FUNCTION_BLOCK QueryServiceOpcUa (* Query for Services using OPC UA *)
  (* Standard: 61499-2; Description: Copyright (c) 2019 fortiss GmbH This program and the accompanying materials are made available under the terms of the Eclipse Public License 2.0 which is available at https://www.eclipse.org/legal/epl-2.0/ SPDX-License-Identifier: EPL-2.0 *)
  (* Version 1.0, 2019-09-17, Jose Cabral, fortiss GmbH *)
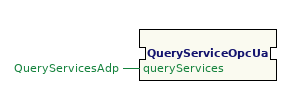
  SOCKETS
    queryServices : QueryServicesAdp;
  END_SOCKETS
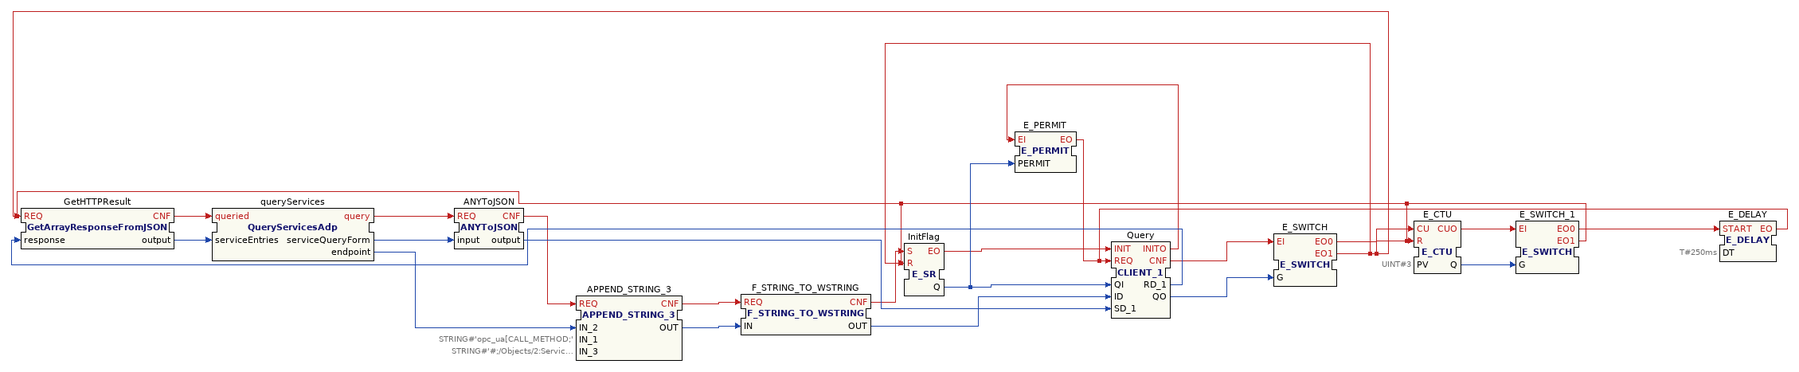
  FBS
    APPEND_STRING_3 : APPEND_STRING_3(IN_1 := STRING#'opc_ua[CALL_METHOD;', IN_3 := STRING#'#;/Objects/2:ServiceRegistry/2:query]');
    F_STRING_TO_WSTRING : F_STRING_TO_WSTRING;
    InitFlag : E_SR;
    E_PERMIT : E_PERMIT;
    ANYToJSON : ANYToJSON;
    GetHTTPResult : GetArrayResponseFromJSON;
    Query : CLIENT_1;
    E_SWITCH_1 : E_SWITCH;
    E_SWITCH : E_SWITCH;
    E_DELAY : E_DELAY(DT := T#250ms);
    E_CTU : E_CTU(PV := UINT#3);
  END_FBS
  EVENT_CONNECTIONS
    APPEND_STRING_3.CNF TO F_STRING_TO_WSTRING.REQ;
    F_STRING_TO_WSTRING.CNF TO InitFlag.S;
    ANYToJSON.CNF TO APPEND_STRING_3.REQ;
    queryServices.query TO ANYToJSON.REQ;
    GetHTTPResult.CNF TO queryServices.queried;
    InitFlag.EO TO Query.INIT;
    E_PERMIT.EO TO Query.REQ;
    Query.INITO TO E_PERMIT.EI;
    E_SWITCH_1.EO0 TO E_DELAY.START;
    E_CTU.CUO TO E_SWITCH_1.EI;
    E_SWITCH.EO0 TO E_CTU.CU;
    E_SWITCH.EO1 TO GetHTTPResult.REQ;
    E_SWITCH.EO1 TO InitFlag.R;
    Query.CNF TO E_SWITCH.EI;
    E_SWITCH_1.EO1 TO InitFlag.R;
    E_SWITCH_1.EO1 TO GetHTTPResult.REQ;
    E_DELAY.EO TO Query.REQ;
    E_SWITCH.EO1 TO E_CTU.R;
    E_SWITCH_1.EO1 TO E_CTU.R;
  END_CONNECTIONS
  DATA_CONNECTIONS
    APPEND_STRING_3.OUT TO F_STRING_TO_WSTRING.IN;
    InitFlag.Q TO E_PERMIT.PERMIT;
    queryServices.serviceQueryForm TO ANYToJSON.input;
    queryServices.endpoint TO APPEND_STRING_3.IN_2;
    GetHTTPResult.output TO queryServices.serviceEntries;
    InitFlag.Q TO Query.QI;
    F_STRING_TO_WSTRING.OUT TO Query.ID;
    ANYToJSON.output TO Query.SD_1;
    Query.RD_1 TO GetHTTPResult.response;
    E_CTU.Q TO E_SWITCH_1.G;
    Query.QO TO E_SWITCH.G;
  END_CONNECTIONS
END_FUNCTION_BLOCK
